# EPICS autosave request: iocs/tpx3IOC/iocBoot/iocTimePix/profiles/mpx3/auto_settings.req
file "ADTimePix_settings.req",  P=$(P),  R=cam1:
file "NDStdArrays_settings.req",  P=$(P),  R=image1:
file "NDStdArrays_settings.req",  P=$(P),  R=imageTh1:
file "NDPva_settings.req",          P=$(P),  R=Pva2:
file "commonPlugin_settings.req", P=$(P)
